FUNCTION CheckRangeSigned : DINT
VAR_INPUT
    value, lower, upper: DINT;
END_VAR
VAR
END_VAR

IF (value < lower) THEN
	CheckRangeSigned_ErrCnt := CheckRangeSigned_ErrCnt + 1;
	CheckRangeSigned := lower;
ELSIF(value > upper) THEN
	CheckRangeSigned_ErrCnt := CheckRangeSigned_ErrCnt + 1;
	CheckRangeSigned := upper;
ELSE
	CheckRangeSigned := value;
END_IF

END_FUNCTION

(* stored: Version 1.1.0.1, ProductVersion 3.1.4024.9
   POU CheckRangeSigned: Id {43d2ac21-bac2-496f-97e4-db04f1b037e5}, SpecialFunc CheckRangeSigned *)
